PROGRAM P_Array_List_Example
VAR
	eState 		: (IDLE, INSERT, REVERSE, RESIZE, GET, SET, FIND, CLEAR, ADD_FRONT, ADD_BACK, REMOVE, REMOVE_AT);
	fbArray_List: FB_Array_List(0);
	nFind 		: DINT;
	sData 		: WSTRING;
	sRTNData	: ARRAY[0..6] OF WSTRING;
	nCount 		: DINT;
	stError 	: ST_ERROR;
END_VAR

stError := fbArray_List._Error_Status;
CASE eState OF
	INSERT:
		sData := "Cats";	fbArray_List.Insert(sData, 0);
		sData := "Dogs";	fbArray_List.Insert(sData, 1);
		sData := "Ravens";	fbArray_List.Insert(sData, 2);
		sData := "Mollies";	fbArray_List.Insert(sData, 3);
	REVERSE:
		fbArray_List.Reverse();
	RESIZE:
		fbArray_List.Resize(3);
	GET: 
		fbArray_List
			.Get(sRTNData[0], 0)
			.Get(sRTNData[1], 1)
			.Get(sRTNData[2], 2)
			.Get(sRTNData[3], 3)
			.Get(sRTNData[4], 4)
			.Get(sRTNData[5], 5)
			.Get(sRTNData[6], 6);
	SET:
		sData := "Ravens";	fbArray_List.Set(sData, 0);
		sData := "Mollies";	fbArray_List.Set(sData, 1);
		sData := "Dogs";	fbArray_List.Set(sData, 2);
		sData := "Cats";	fbArray_List.Set(sData, 3);
	FIND:
		sData := "Dogs"; fbArray_List.Find(sData, nIndex => nFind);
	CLEAR:
		fbArray_List.Clear();
	ADD_FRONT:
		sData := "Pythons";fbArray_List.Add_Front(sData);
	ADD_BACK:
		sData := "Anacondas"; fbArray_List.Add_Back(sData);
	REMOVE:
		fbArray_List.Remove();
	REMOVE_AT:
		fbArray_List.RemoveAt(2);
END_CASE
nCount := fbArray_List._Count;
eState := IDLE;

END_PROGRAM

(* stored: Version 1.1.0.1, ProductVersion 3.1.4024.4
   POU P_Array_List_Example: Id {969256da-a7e7-43a9-8f8a-e825c77e7067}, SpecialFunc None *)
